//LREAL average filter
FUNCTION_BLOCK AverageFilter
VAR_INPUT	
	IN														: LREAL;		// Adds value for average calculation
END_VAR
VAR_OUTPUT
	Q														: LREAL:=0.0;	// Result of average calculation
	Valid													: BOOL:=FALSE;	// Is TRUE once a value is inserted
END_VAR         											
VAR             											
	Total													: LREAL:=0.0;
	Count													: LREAL:=0;
END_VAR

Insert(IN);

METHOD PUBLIC clear : booL; //Return value = TRUE if execution finished
VAR_INPUT
END_VAR
Q:=Total	:=0.0;
Valid		:=FALSE;
Count		:=0.0;
Clear		:= TRUE;
END_METHOD

METHOD PUBLIC insert : LREAL //Result = actual average value
VAR_INPUT
	Value								:	LREAL ;
END_VAR
Total		:=Total+Value;
Count		:=Count+1.0;
Q			:=Total/Count;
Valid		:=TRUE;
Insert 		:= Q;
END_METHOD

END_FUNCTION_BLOCK

(* stored: Version 1.1.0.1, ProductVersion 3.1.4024.3
   POU AverageFilter: Id {48cfc97c-e9b1-41f1-ba51-69be3fe79492}, SpecialFunc None
   Method clear: Id {65255996-d613-4b5c-8168-5ad802a98d02}
   Method insert: Id {c7f0bd30-a4a0-40e3-a4b5-6e8af2e34e9e} *)
